(* PLC project pequenaFabrica5.project, CODESYS CODESYS V3.5 SP16 Patch 3 *)
(* stored: creationDateTime 2021-09-05T20:49:14.5976402, modificationDateTime 2021-07-19T00:15:29.4418959 *)

PROGRAM sfcM1

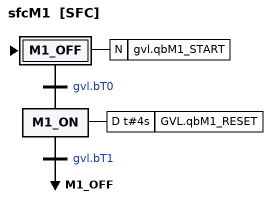
INITIAL_STEP M1_OFF:
  gvl.qbM1_START(N);
END_STEP
TRANSITION FROM M1_OFF TO M1_ON
  := gvl.bT0;
END_TRANSITION
STEP M1_ON:
  GVL.qbM1_RESET(D, t#4s);
END_STEP
TRANSITION FROM M1_ON TO M1_OFF
  := gvl.bT1;
END_TRANSITION
END_PROGRAM

PROGRAM sfcM2

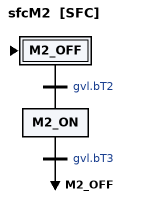
INITIAL_STEP M2_OFF:
END_STEP
TRANSITION FROM M2_OFF TO M2_ON
  := gvl.bT2;
END_TRANSITION
STEP M2_ON:
END_STEP
TRANSITION FROM M2_ON TO M2_OFF
  := gvl.bT3;
END_TRANSITION
END_PROGRAM

PROGRAM sfcBUFFER

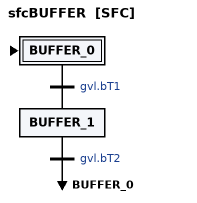
INITIAL_STEP BUFFER_0:
END_STEP
TRANSITION FROM BUFFER_0 TO BUFFER_1
  := gvl.bT1;
END_TRANSITION
STEP BUFFER_1:
END_STEP
TRANSITION FROM BUFFER_1 TO BUFFER_0
  := gvl.bT2;
END_TRANSITION
END_PROGRAM

PROGRAM sfcAUTONET

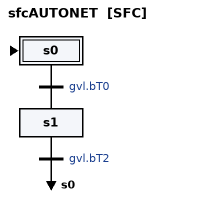
INITIAL_STEP s0:
END_STEP
TRANSITION FROM s0 TO s1
  := gvl.bT0;
END_TRANSITION
STEP s1:
END_STEP
TRANSITION FROM s1 TO s0
  := gvl.bT2;
END_TRANSITION
END_PROGRAM

PROGRAM stTransitions

                  
gvl.bT0:= sfcM1.M1_OFF.x AND sfcAUTONET.s0.x AND GVL.qbM1_START;

GVL.RTRIG1(CLK:=GVL.ibM1_END);
gvl.bT1:= sfcM1.M1_ON.x AND GVL.RTRIG1.Q;

gvl.bT2:= sfcM2.M2_OFF.x AND sfcAUTONET.s1.x AND sfcBUFFER.BUFFER_1.x AND GVL.qbM2_START;

GVL.RTRIG3(CLK:=gvl.ibM2_END);
gvl.bT3:= sfcM2.M2_ON.x AND GVL.RTRIG3.Q;
                
END_PROGRAM

CONFIGURATION Application
  RESOURCE Application ON PLC
    {attribute 'qualified_only'}
    VAR_GLOBAL  (* GVL *)
      qbM1_START : BOOL;
      qbM2_START : BOOL;
      ibM1_END : BOOL;
      ibM2_END : BOOL;
      RTRIG1 : R_TRIG;
      RTRIG2 : R_TRIG;
      RTRIG3 : R_TRIG;
      RTRIG4 : R_TRIG;
      bT0 : BOOL;
      bT1 : BOOL;
      bT2 : BOOL;
      bT3 : BOOL;
      qbM1_RESET : BOOL;
    END_VAR
    TASK MainTask(INTERVAL := T#50ms, PRIORITY := 0);
    PROGRAM sfcM1 WITH MainTask : sfcM1;
    PROGRAM sfcM2 WITH MainTask : sfcM2;
    PROGRAM sfcBUFFER WITH MainTask : sfcBUFFER;
    PROGRAM sfcAUTONET WITH MainTask : sfcAUTONET;
    PROGRAM stTransitions WITH MainTask : stTransitions;
  END_RESOURCE
END_CONFIGURATION
